Universal Robots PolyScope program: cable_extend_v3.urp

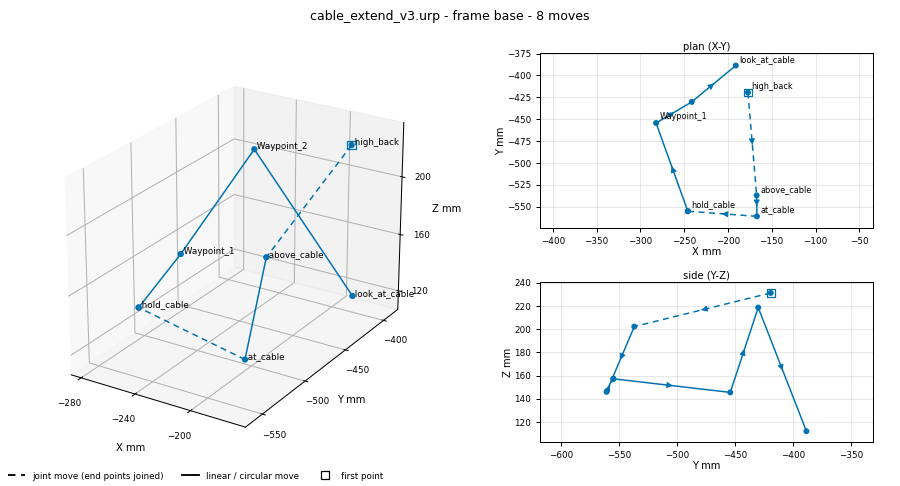
[picture p0: tool path of cable_extend_v3.urp in frame base, 8 of 8 moves have a stored position in this frame; points joined in program order, loops and branches not executed]
Program cable_extend_v3 (installation=default directory=/programs/wrs2020 createdIn=3.8.0.61336 lastSavedIn=5.10.0.106288 robotSerialNumber=20205500607)
Calibrated DH parameters: a=[0.000096, -0.337, -0.383372, 0.000118, 0.000015, 0]; d=[0.162724, 79.377998, -95.545185, 16.300583, 0.099689, 0.099499]; alpha=[1.569249, 0.003272, 0.005201, 1.570041, -1.570219, 0]; deltaTheta=[0, 0.65664, 5.410619, 0.215927, -0.000001, 0]
Robot Program (runOnlyOnce=true)
  Popup Message (haltProgram=false message=wait for a_bot to prepare cable inputType=Text)
  URCap Gripper (Robotiq_Grippers, Robotiq Inc.) dataModel(position=72.15686274509804, force=100.0, speed=100.0, positionInDouble=72.15686274509804, forceInDouble=100.0, speedInDouble=100.0, slaveIds=[9], blocking=true)
  MoveJ speed 60 deg/s, acceleration 80 deg/s^2 (useActiveTCP=false) tcp=gripper_85_tip; feature=Base
    Waypoint high_back: TCP in base x=-177.128 y=-419.476 z=231.31 mm, rx=2.059 ry=-1.9344 rz=0.3994 rad; joints [39.252, -108.249, 125.554, -122.083, -71.876, 217.968] deg; TCP offset x=0 y=0 z=165 mm, rx=0 ry=0 rz=0 rad
    Waypoint above_cable: TCP in base x=-167.206 y=-537.006 z=202.342 mm, rx=2.059 ry=-1.9344 rz=0.3994 rad; joints [52.264, -90.132, 116.291, -134.547, -75.59, 231.045] deg
  MoveL speed 100 mm/s, acceleration 200 mm/s^2 (useActiveTCP=false) tcp=gripper_85_tip; feature=Base
    Waypoint at_cable: TCP in base x=-166.902 y=-560.898 z=146.118 mm, rx=2.0589 ry=-1.9344 rz=0.3994 rad; joints [54.065, -82.676, 117.922, -144.07, -76.183, 232.868] deg
  URCap Gripper (Robotiq_Grippers, Robotiq Inc.) dataModel(position=85.09803921568627, force=100.0, speed=0.0, positionInDouble=85.09803921568627, forceInDouble=100.0, speedInDouble=0.0, slaveIds=[9], blocking=true)
  Popup Message (haltProgram=false message=wait for a_bot to release inputType=Text)
  MoveL speed 10 mm/s, acceleration 250 mm/s^2 (useActiveTCP=false) tcp=gripper_85_tip; feature=Base
    MoveDirectionNode (selectedDirection=XMinus)
      Until DISTANCE (allowActions=false deceleration=3 distanceNodeType=STOP) Distance=0.129; motionParameters(blendRadius=0)
  URCap Gripper (Robotiq_Grippers, Robotiq Inc.) dataModel(position=100.0, force=100.0, speed=100.0, positionInDouble=100.0, forceInDouble=100.0, speedInDouble=100.0, slaveIds=[9], blocking=true)
  MoveJ speed 60 deg/s, acceleration 80 deg/s^2 (useActiveTCP=false) tcp=gripper_85_tip; feature=Base
    Waypoint hold_cable: TCP in base x=-245.776 y=-555.018 z=157.329 mm, rx=0.8037 ry=-2.5295 rz=1.1507 rad; joints [37.455, -78.709, 129.699, -175.898, -52.973, 284.397] deg
    SuppressedNode
      Waypoint Waypoint_5: TCP in base x=-282.891 y=-437.459 z=279.407 mm, rx=0.0863 ry=-2.8917 rz=1.1802 rad; joints [39.548, -82.252, 116.923, -156.05, -57.537, 315.725] deg; TCP offset x=0 y=0 z=0 mm, rx=0 ry=0 rz=0 rad
  Popup Message (haltProgram=false message=wait for a_bot to grasp cable. press enter to straighten cable and go observe inputType=Text)
  Loop Counting (count=3) loopVariable(name=Loop_1)
    MoveL speed 250 mm/s, acceleration 1200 mm/s^2 (useActiveTCP=true) feature=Base
      Waypoint hold_cable: TCP in base x=-245.776 y=-555.018 z=157.329 mm, rx=0.8037 ry=-2.5295 rz=1.1507 rad; joints [37.455, -78.709, 129.699, -175.898, -52.973, 284.397] deg; TCP offset x=0 y=0 z=165 mm, rx=0 ry=0 rz=0 rad
      URCap Gripper (Robotiq_Grippers, Robotiq Inc.) dataModel(position=100.0, force=0.0, speed=100.0, positionInDouble=100.0, forceInDouble=0.0, speedInDouble=100.0, slaveIds=[9], blocking=true)
      MoveDirectionNode (selectedDirection=YPlus toolParams=0.01, 0.2) feature=Joint_6_name
        Until DISTANCE (allowActions=false deceleration=3 distanceNodeType=STOP) Distance=0.012; motionParameters(blendRadius=0)
      URCap Gripper (Robotiq_Grippers, Robotiq Inc.) dataModel(position=48.627450980392155, force=0.0, speed=100.0, positionInDouble=48.627450980392155, forceInDouble=0.0, speedInDouble=100.0, slaveIds=[9], blocking=true)
      SuppressedNode
        Waypoint pull_start: TCP in base x=-256.402 y=-559.701 z=148.507 mm, rx=-0.0406 ry=2.8584 rz=-1.2945 rad; joints [36.887, -76.525, 128.286, -175.624, -52.262, 317.319] deg
  URCap Gripper (Robotiq_Grippers, Robotiq Inc.) dataModel(position=0.0, force=100.0, speed=100.0, positionInDouble=0.0, forceInDouble=100.0, speedInDouble=100.0, slaveIds=[9], blocking=true)
  MoveL speed 250 mm/s, acceleration 1200 mm/s^2 (useActiveTCP=false) tcp=gripper_85_tip; feature=Base
    Waypoint Waypoint_1: TCP in base x=-282.011 y=-454.343 z=145.637 mm, rx=0.0882 ry=-2.9758 rz=0.9624 rad; joints [27.873, -89.876, 131.134, -149.666, -58.399, 299.802] deg
    Waypoint Waypoint_2: TCP in base x=-241.284 y=-430.243 z=218.721 mm, rx=0.0882 ry=-2.9758 rz=0.9624 rad; joints [27.542, -104.305, 130.323, -134.175, -58.276, 299.32] deg
    Waypoint look_at_cable: TCP in base x=-191.011 y=-388.704 z=112.194 mm, rx=-0.0175 ry=-3.0299 rz=0.8172 rad; joints [28.911, -103.299, 145.338, -148.082, -63.832, 303.371] deg
